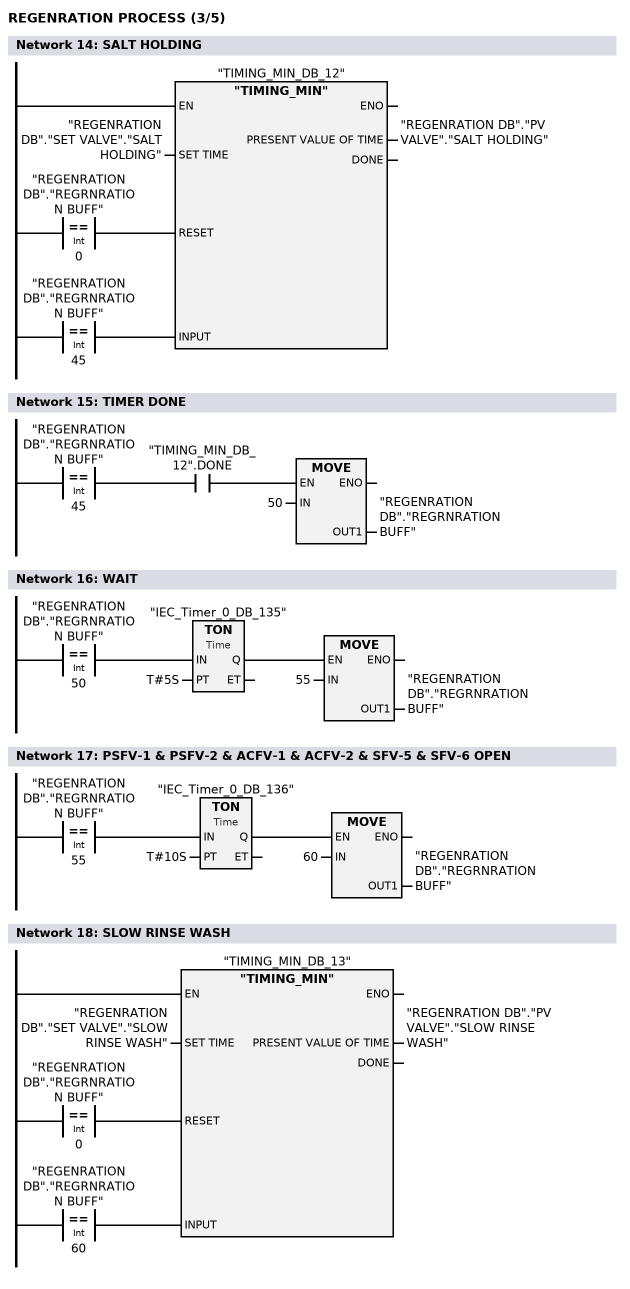
   RUNG wire#powerrail
      "TIMING_MIN_DB_12"(RESET := wire#w1, INPUT := wire#w2, "SET TIME" := "REGENRATION DB"."SET VALVE"."SALT HOLDING", "PRESENT VALUE OF TIME" => "REGENRATION DB"."PV VALVE"."SALT HOLDING", DONE =>)
   END_RUNG
   RUNG wire#powerrail
      { S7_Templates := "SrcType := Int" } EQ_Contact(in1 := "REGENRATION DB"."REGRNRATION BUFF", in2 := 0)
   END_RUNG wire#w1
   RUNG wire#powerrail
      { S7_Templates := "SrcType := Int" } EQ_Contact(in1 := "REGENRATION DB"."REGRNRATION BUFF", in2 := 45)
   END_RUNG wire#w2
   // the same network as SCL:
   "TIMING_MIN_DB_12"("SET TIME" := "REGENRATION DB"."SET VALVE"."SALT HOLDING",   // "TIMING_MIN"
                      RESET := "REGENRATION DB"."REGRNRATION BUFF" = 0,
                      INPUT := "REGENRATION DB"."REGRNRATION BUFF" = 45,
                      "PRESENT VALUE OF TIME" => "REGENRATION DB"."PV VALVE"."SALT HOLDING");
END_REGION

REGION Network 15: TIMER DONE
   RUNG wire#powerrail
      { S7_Templates := "SrcType := Int" } EQ_Contact(in1 := "REGENRATION DB"."REGRNRATION BUFF", in2 := 45)
      Contact( "TIMING_MIN_DB_12".DONE )
      Move(in := 50, out1 => "REGENRATION DB"."REGRNRATION BUFF")
   END_RUNG
   // the same network as SCL:
   IF ("REGENRATION DB"."REGRNRATION BUFF" = 45) AND "TIMING_MIN_DB_12".DONE THEN
       "REGENRATION DB"."REGRNRATION BUFF" := 50;
   END_IF;
END_REGION

REGION Network 16: WAIT
   RUNG wire#powerrail
      { S7_Templates := "SrcType := Int" } EQ_Contact(in1 := "REGENRATION DB"."REGRNRATION BUFF", in2 := 50)
      { S7_Templates := "time_type := Time" } "IEC_Timer_0_DB_135".TON(pt := T#5S, et =>)
      Move(in := 55, out1 => "REGENRATION DB"."REGRNRATION BUFF")
   END_RUNG
   // the same network as SCL:
   "IEC_Timer_0_DB_135".TON(IN := "REGENRATION DB"."REGRNRATION BUFF" = 50, PT := T#5S);
   IF "IEC_Timer_0_DB_135".Q THEN "REGENRATION DB"."REGRNRATION BUFF" := 55; END_IF;
END_REGION

REGION Network 17: PSFV-1 & PSFV-2 & ACFV-1 & ACFV-2 & SFV-5 & SFV-6 OPEN
   RUNG wire#powerrail
      { S7_Templates := "SrcType := Int" } EQ_Contact(in1 := "REGENRATION DB"."REGRNRATION BUFF", in2 := 55)
      { S7_Templates := "time_type := Time" } "IEC_Timer_0_DB_136".TON(pt := T#10S, et =>)
      Move(in := 60, out1 => "REGENRATION DB"."REGRNRATION BUFF")
   END_RUNG
   // the same network as SCL:
   "IEC_Timer_0_DB_136".TON(IN := "REGENRATION DB"."REGRNRATION BUFF" = 55, PT := T#10S);
   IF "IEC_Timer_0_DB_136".Q THEN "REGENRATION DB"."REGRNRATION BUFF" := 60; END_IF;
END_REGION

REGION Network 18: SLOW RINSE WASH
   RUNG wire#powerrail
      "TIMING_MIN_DB_13"(RESET := wire#w1, INPUT := wire#w2, "SET TIME" := "REGENRATION DB"."SET VALVE"."SLOW RINSE WASH", "PRESENT VALUE OF TIME" => "REGENRATION DB"."PV VALVE"."SLOW RINSE WASH", DONE =>)
   END_RUNG
   RUNG wire#powerrail
      { S7_Templates := "SrcType := Int" } EQ_Contact(in1 := "REGENRATION DB"."REGRNRATION BUFF", in2 := 0)
   END_RUNG wire#w1
   RUNG wire#powerrail
      { S7_Templates := "SrcType := Int" } EQ_Contact(in1 := "REGENRATION DB"."REGRNRATION BUFF", in2 := 60)
   END_RUNG wire#w2
   // the same network as SCL:
   "TIMING_MIN_DB_13"("SET TIME" := "REGENRATION DB"."SET VALVE"."SLOW RINSE WASH",   // "TIMING_MIN"
                      RESET := "REGENRATION DB"."REGRNRATION BUFF" = 0,
                      INPUT := "REGENRATION DB"."REGRNRATION BUFF" = 60,
                      "PRESENT VALUE OF TIME" => "REGENRATION DB"."PV VALVE"."SLOW RINSE WASH");
END_REGION

REGION Network 19: TIMER DONE
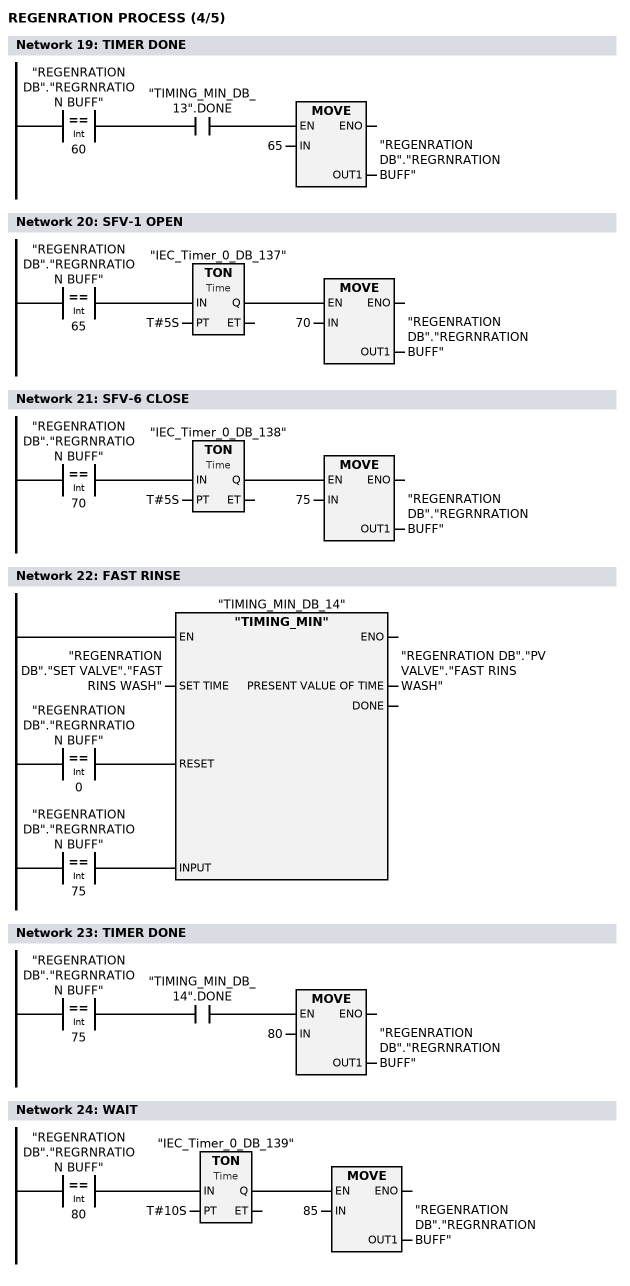
   RUNG wire#powerrail
      { S7_Templates := "SrcType := Int" } EQ_Contact(in1 := "REGENRATION DB"."REGRNRATION BUFF", in2 := 60)
      Contact( "TIMING_MIN_DB_13".DONE )
      Move(in := 65, out1 => "REGENRATION DB"."REGRNRATION BUFF")
   END_RUNG
   // the same network as SCL:
   IF ("REGENRATION DB"."REGRNRATION BUFF" = 60) AND "TIMING_MIN_DB_13".DONE THEN
       "REGENRATION DB"."REGRNRATION BUFF" := 65;
   END_IF;
END_REGION

REGION Network 20: SFV-1 OPEN
   RUNG wire#powerrail
      { S7_Templates := "SrcType := Int" } EQ_Contact(in1 := "REGENRATION DB"."REGRNRATION BUFF", in2 := 65)
      { S7_Templates := "time_type := Time" } "IEC_Timer_0_DB_137".TON(pt := T#5S, et =>)
      Move(in := 70, out1 => "REGENRATION DB"."REGRNRATION BUFF")
   END_RUNG
   // the same network as SCL:
   "IEC_Timer_0_DB_137".TON(IN := "REGENRATION DB"."REGRNRATION BUFF" = 65, PT := T#5S);
   IF "IEC_Timer_0_DB_137".Q THEN "REGENRATION DB"."REGRNRATION BUFF" := 70; END_IF;
END_REGION

REGION Network 21: SFV-6 CLOSE
   RUNG wire#powerrail
      { S7_Templates := "SrcType := Int" } EQ_Contact(in1 := "REGENRATION DB"."REGRNRATION BUFF", in2 := 70)
      { S7_Templates := "time_type := Time" } "IEC_Timer_0_DB_138".TON(pt := T#5S, et =>)
      Move(in := 75, out1 => "REGENRATION DB"."REGRNRATION BUFF")
   END_RUNG
   // the same network as SCL:
   "IEC_Timer_0_DB_138".TON(IN := "REGENRATION DB"."REGRNRATION BUFF" = 70, PT := T#5S);
   IF "IEC_Timer_0_DB_138".Q THEN "REGENRATION DB"."REGRNRATION BUFF" := 75; END_IF;
END_REGION

REGION Network 22: FAST RINSE
   RUNG wire#powerrail
      "TIMING_MIN_DB_14"(RESET := wire#w1, INPUT := wire#w2, "SET TIME" := "REGENRATION DB"."SET VALVE"."FAST RINS WASH", "PRESENT VALUE OF TIME" => "REGENRATION DB"."PV VALVE"."FAST RINS WASH", DONE =>)
   END_RUNG
   RUNG wire#powerrail
      { S7_Templates := "SrcType := Int" } EQ_Contact(in1 := "REGENRATION DB"."REGRNRATION BUFF", in2 := 0)
   END_RUNG wire#w1
   RUNG wire#powerrail
      { S7_Templates := "SrcType := Int" } EQ_Contact(in1 := "REGENRATION DB"."REGRNRATION BUFF", in2 := 75)
   END_RUNG wire#w2
   // the same network as SCL:
   "TIMING_MIN_DB_14"("SET TIME" := "REGENRATION DB"."SET VALVE"."FAST RINS WASH",   // "TIMING_MIN"
                      RESET := "REGENRATION DB"."REGRNRATION BUFF" = 0,
                      INPUT := "REGENRATION DB"."REGRNRATION BUFF" = 75,
                      "PRESENT VALUE OF TIME" => "REGENRATION DB"."PV VALVE"."FAST RINS WASH");
END_REGION

REGION Network 23: TIMER DONE
   RUNG wire#powerrail
      { S7_Templates := "SrcType := Int" } EQ_Contact(in1 := "REGENRATION DB"."REGRNRATION BUFF", in2 := 75)
      Contact( "TIMING_MIN_DB_14".DONE )
      Move(in := 80, out1 => "REGENRATION DB"."REGRNRATION BUFF")
   END_RUNG
   // the same network as SCL:
   IF ("REGENRATION DB"."REGRNRATION BUFF" = 75) AND "TIMING_MIN_DB_14".DONE THEN
       "REGENRATION DB"."REGRNRATION BUFF" := 80;
   END_IF;
END_REGION

REGION Network 24: WAIT
   RUNG wire#powerrail
      { S7_Templates := "SrcType := Int" } EQ_Contact(in1 := "REGENRATION DB"."REGRNRATION BUFF", in2 := 80)
      { S7_Templates := "time_type := Time" } "IEC_Timer_0_DB_139".TON(pt := T#10S, et =>)
      Move(in := 85, out1 => "REGENRATION DB"."REGRNRATION BUFF")
   END_RUNG
   // the same network as SCL:
   "IEC_Timer_0_DB_139".TON(IN := "REGENRATION DB"."REGRNRATION BUFF" = 80, PT := T#10S);
   IF "IEC_Timer_0_DB_139".Q THEN "REGENRATION DB"."REGRNRATION BUFF" := 85; END_IF;
END_REGION

REGION Network 25: PSFV-1 & PSFV-2 & ACFV-1 & ACFV-2 & SFV-5 & SFV-1 CLOSE
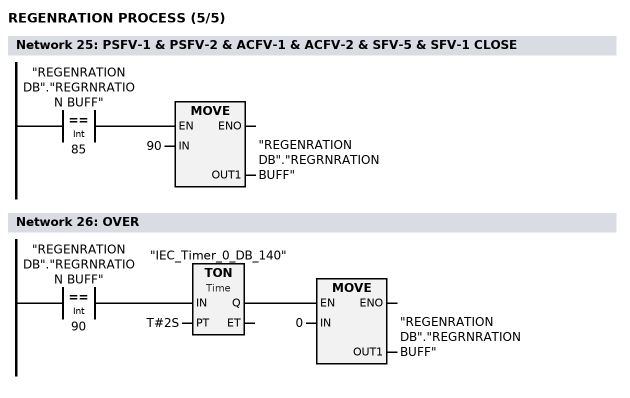
   RUNG wire#powerrail
      { S7_Templates := "SrcType := Int" } EQ_Contact(in1 := "REGENRATION DB"."REGRNRATION BUFF", in2 := 85)
      Move(in := 90, out1 => "REGENRATION DB"."REGRNRATION BUFF")
   END_RUNG
   // the same network as SCL:
   IF "REGENRATION DB"."REGRNRATION BUFF" = 85 THEN "REGENRATION DB"."REGRNRATION BUFF" := 90; END_IF;
END_REGION

REGION Network 26: OVER
   RUNG wire#powerrail
      { S7_Templates := "SrcType := Int" } EQ_Contact(in1 := "REGENRATION DB"."REGRNRATION BUFF", in2 := 90)
      { S7_Templates := "time_type := Time" } "IEC_Timer_0_DB_140".TON(pt := T#2S, et =>)
      Move(in := 0, out1 => "REGENRATION DB"."REGRNRATION BUFF")
   END_RUNG
   // the same network as SCL:
   "IEC_Timer_0_DB_140".TON(IN := "REGENRATION DB"."REGRNRATION BUFF" = 90, PT := T#2S);
   IF "IEC_Timer_0_DB_140".Q THEN "REGENRATION DB"."REGRNRATION BUFF" := 0; END_IF;
END_REGION
END_FUNCTION

FUNCTION "RO PROCESS." : Void   // FC15, LAD
{ S7_Optimized_Access := 'TRUE' }
// stored: SetENOAutomatically false
BEGIN

REGION Network 1: AUTO FLUSHING AV3
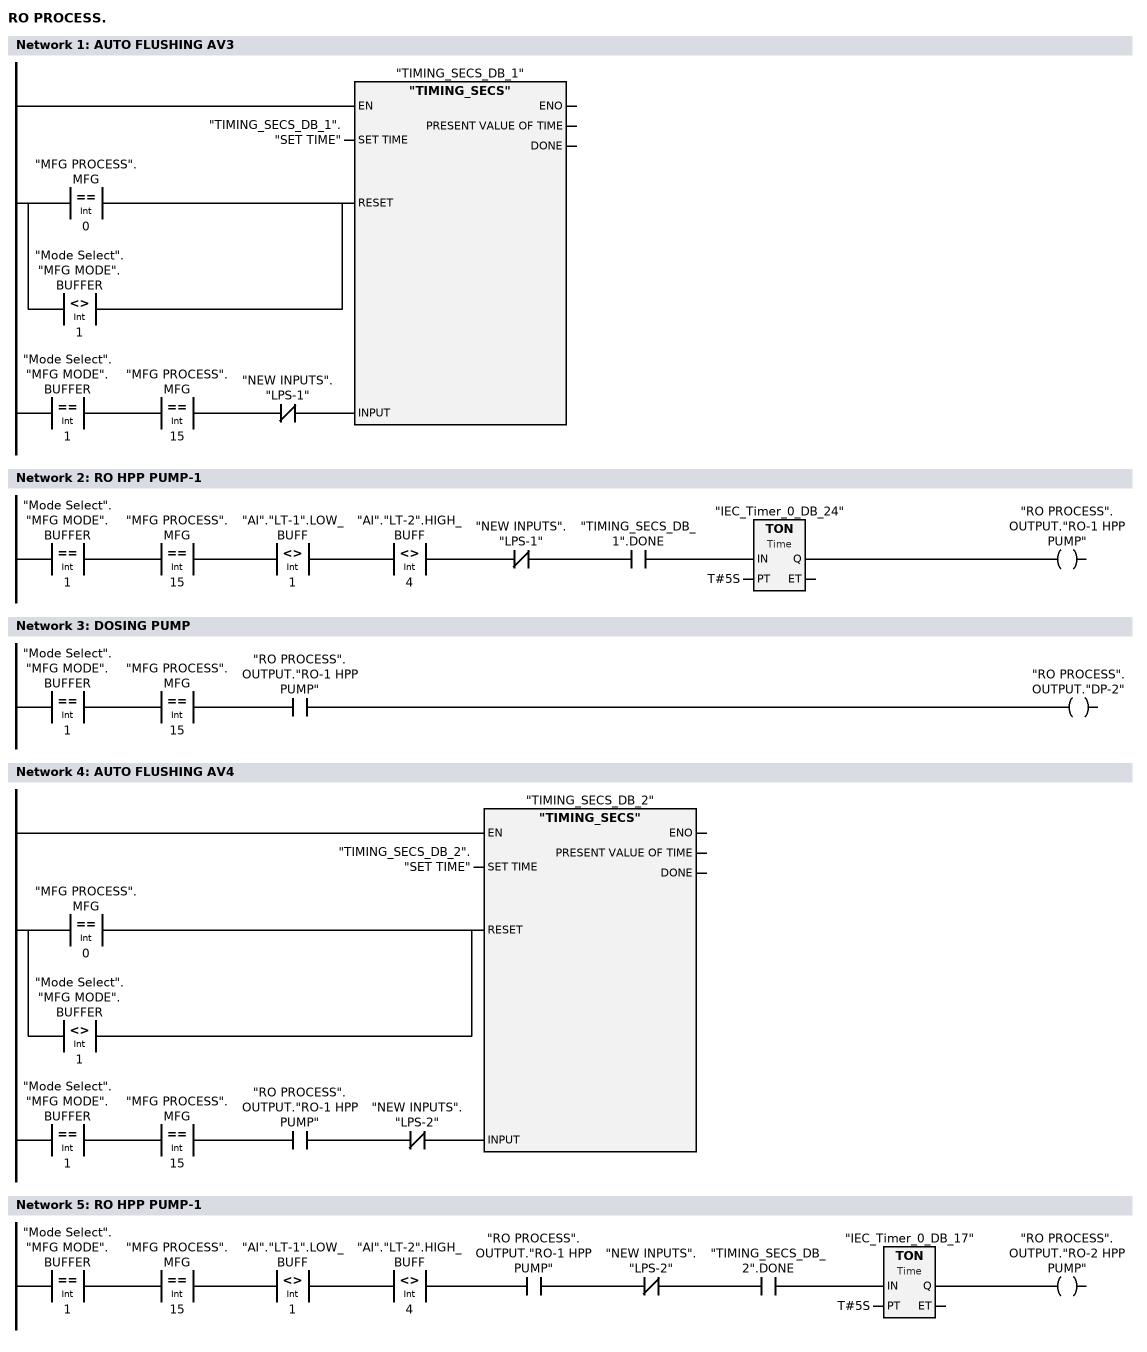
   RUNG wire#powerrail
      "TIMING_SECS_DB_1"(RESET := wire#w1, INPUT := wire#w2, "SET TIME" := "TIMING_SECS_DB_1"."SET TIME", "PRESENT VALUE OF TIME" =>, DONE =>)
   END_RUNG
   RUNG wire#powerrail
      { S7_Templates := "SrcType := Int" } EQ_Contact(in1 := "MFG PROCESS".MFG, in2 := 0)
   END_RUNG wire#w1
   RUNG wire#powerrail
      { S7_Templates := "SrcType := Int" } NE_Contact(in1 := "Mode Select"."MFG MODE".BUFFER, in2 := 1)
   END_RUNG wire#w1
   RUNG wire#powerrail
      { S7_Templates := "SrcType := Int" } EQ_Contact(in1 := "Mode Select"."MFG MODE".BUFFER, in2 := 1)
      { S7_Templates := "SrcType := Int" } EQ_Contact(in1 := "MFG PROCESS".MFG, in2 := 15)
      I_Contact( "NEW INPUTS"."LPS-1" )
   END_RUNG wire#w2
   // the same network as SCL:
   "TIMING_SECS_DB_1"("SET TIME" := "TIMING_SECS_DB_1"."SET TIME",   // "TIMING_SECS"
                      RESET := ("MFG PROCESS".MFG = 0) OR ("Mode Select"."MFG MODE".BUFFER <> 1),
                      INPUT := ("Mode Select"."MFG MODE".BUFFER = 1) AND ("MFG PROCESS".MFG = 15) AND NOT "NEW INPUTS"."LPS-1");
END_REGION

REGION Network 2: RO HPP PUMP-1
   RUNG wire#powerrail
      { S7_Templates := "SrcType := Int" } EQ_Contact(in1 := "Mode Select"."MFG MODE".BUFFER, in2 := 1)
      { S7_Templates := "SrcType := Int" } EQ_Contact(in1 := "MFG PROCESS".MFG, in2 := 15)
      { S7_Templates := "SrcType := Int" } NE_Contact(in1 := "AI"."LT-1".LOW_BUFF, in2 := 1)
      { S7_Templates := "SrcType := Int" } NE_Contact(in1 := "AI"."LT-2".HIGH_BUFF, in2 := 4)
      I_Contact( "NEW INPUTS"."LPS-1" )
      Contact( "TIMING_SECS_DB_1".DONE )
      { S7_Templates := "time_type := Time" } "IEC_Timer_0_DB_24".TON(pt := T#5S, et =>)
      Coil( "RO PROCESS".OUTPUT."RO-1 HPP PUMP" )
   END_RUNG
   // the same network as SCL:
   "IEC_Timer_0_DB_24".TON(IN := ("Mode Select"."MFG MODE".BUFFER = 1) AND ("MFG PROCESS".MFG = 15) AND ("AI"."LT-1".LOW_BUFF <> 1) AND ("AI"."LT-2".HIGH_BUFF <> 4) AND NOT "NEW INPUTS"."LPS-1" AND "TIMING_SECS_DB_1".DONE,
                           PT := T#5S);
   "RO PROCESS".OUTPUT."RO-1 HPP PUMP" := "IEC_Timer_0_DB_24".Q;
END_REGION

REGION Network 3: DOSING PUMP
   RUNG wire#powerrail
      { S7_Templates := "SrcType := Int" } EQ_Contact(in1 := "Mode Select"."MFG MODE".BUFFER, in2 := 1)
      { S7_Templates := "SrcType := Int" } EQ_Contact(in1 := "MFG PROCESS".MFG, in2 := 15)
      Contact( "RO PROCESS".OUTPUT."RO-1 HPP PUMP" )
      Coil( "RO PROCESS".OUTPUT."DP-2" )
   END_RUNG
   // the same network as SCL:
   "RO PROCESS".OUTPUT."DP-2" := ("Mode Select"."MFG MODE".BUFFER = 1) AND ("MFG PROCESS".MFG = 15) AND "RO PROCESS".OUTPUT."RO-1 HPP PUMP";
END_REGION

REGION Network 4: AUTO FLUSHING AV4
   RUNG wire#powerrail
      "TIMING_SECS_DB_2"(RESET := wire#w1, INPUT := wire#w2, "SET TIME" := "TIMING_SECS_DB_2"."SET TIME", "PRESENT VALUE OF TIME" =>, DONE =>)
   END_RUNG
   RUNG wire#powerrail
      { S7_Templates := "SrcType := Int" } EQ_Contact(in1 := "MFG PROCESS".MFG, in2 := 0)
   END_RUNG wire#w1
   RUNG wire#powerrail
      { S7_Templates := "SrcType := Int" } NE_Contact(in1 := "Mode Select"."MFG MODE".BUFFER, in2 := 1)
   END_RUNG wire#w1
   RUNG wire#powerrail
      { S7_Templates := "SrcType := Int" } EQ_Contact(in1 := "Mode Select"."MFG MODE".BUFFER, in2 := 1)
      { S7_Templates := "SrcType := Int" } EQ_Contact(in1 := "MFG PROCESS".MFG, in2 := 15)
      Contact( "RO PROCESS".OUTPUT."RO-1 HPP PUMP" )
      I_Contact( "NEW INPUTS"."LPS-2" )
   END_RUNG wire#w2
   // the same network as SCL:
   "TIMING_SECS_DB_2"("SET TIME" := "TIMING_SECS_DB_2"."SET TIME",   // "TIMING_SECS"
                      RESET := ("MFG PROCESS".MFG = 0) OR ("Mode Select"."MFG MODE".BUFFER <> 1),
                      INPUT := ("Mode Select"."MFG MODE".BUFFER = 1) AND ("MFG PROCESS".MFG = 15) AND "RO PROCESS".OUTPUT."RO-1 HPP PUMP" AND NOT "NEW INPUTS"."LPS-2");
END_REGION

REGION Network 5: RO HPP PUMP-1
   RUNG wire#powerrail
      { S7_Templates := "SrcType := Int" } EQ_Contact(in1 := "Mode Select"."MFG MODE".BUFFER, in2 := 1)
      { S7_Templates := "SrcType := Int" } EQ_Contact(in1 := "MFG PROCESS".MFG, in2 := 15)
      { S7_Templates := "SrcType := Int" } NE_Contact(in1 := "AI"."LT-1".LOW_BUFF, in2 := 1)
      { S7_Templates := "SrcType := Int" } NE_Contact(in1 := "AI"."LT-2".HIGH_BUFF, in2 := 4)
      Contact( "RO PROCESS".OUTPUT."RO-1 HPP PUMP" )
      I_Contact( "NEW INPUTS"."LPS-2" )
      Contact( "TIMING_SECS_DB_2".DONE )
      { S7_Templates := "time_type := Time" } "IEC_Timer_0_DB_17".TON(pt := T#5S, et =>)
      Coil( "RO PROCESS".OUTPUT."RO-2 HPP PUMP" )
   END_RUNG
   // the same network as SCL:
   "IEC_Timer_0_DB_17".TON(IN := ("Mode Select"."MFG MODE".BUFFER = 1) AND ("MFG PROCESS".MFG = 15) AND ("AI"."LT-1".LOW_BUFF <> 1) AND ("AI"."LT-2".HIGH_BUFF <> 4) AND "RO PROCESS".OUTPUT."RO-1 HPP PUMP" AND NOT "NEW INPUTS"."LPS-2" AND "TIMING_SECS_DB_2".DONE,
                           PT := T#5S);
   "RO PROCESS".OUTPUT."RO-2 HPP PUMP" := "IEC_Timer_0_DB_17".Q;
END_REGION
END_FUNCTION

FUNCTION_BLOCK "TIMING_SECS"   // FB1, LAD
{ S7_Optimized_Access := 'TRUE' }
// stored: MemoryReserve 100, SetENOAutomatically false
   VAR_INPUT
      "SET TIME" : Int;
      RESET : Bool;
      INPUT : Bool;
   END_VAR
   VAR_OUTPUT
      "PRESENT VALUE OF TIME" : Int;
      DONE : Bool;
   END_VAR
   VAR
      "TIMER 1" { S7_SetPoint := 'True'} : IEC_TIMER;
   END_VAR
   VAR RETAIN
      "COUNTER1 1" { S7_SetPoint := 'True'} : IEC_COUNTER;
   END_VAR
   VAR_TEMP   // added for the SCL form of the ladder/FBD networks
      _w1 : Bool;
      _w2 : Bool;
   END_VAR
BEGIN

REGION Network 1
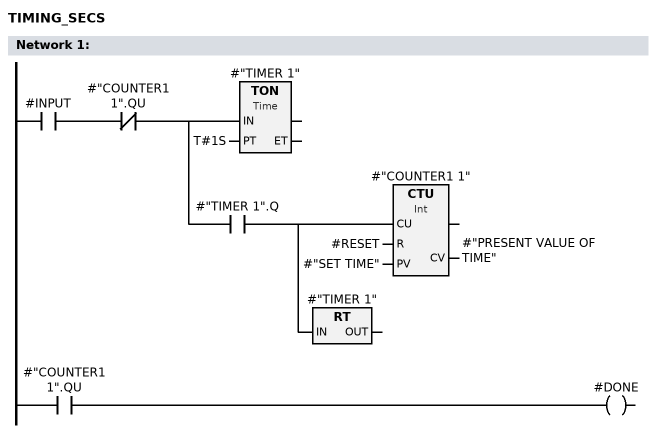
   RUNG wire#powerrail
      Contact( #INPUT )
      I_Contact( #"COUNTER1 1".QU )
      wire#w1
      { S7_Templates := "time_type := Time" } #"TIMER 1".TON(pt := T#1S, et =>)
   END_RUNG
   RUNG wire#w1
      Contact( #"TIMER 1".Q )
      wire#w2
      { S7_Templates := "value_type := Int" } #"COUNTER1 1".CTU(r := #RESET, pv := #"SET TIME", cv => #"PRESENT VALUE OF TIME")
   END_RUNG
   RUNG wire#w2
      RT_Coil( #"TIMER 1" )
   END_RUNG
   RUNG wire#powerrail
      Contact( #"COUNTER1 1".QU )
      Coil( #DONE )
   END_RUNG
   // the same network as SCL:
   #_w1 := #INPUT AND NOT #"COUNTER1 1".QU;
   #"TIMER 1".TON(IN := #_w1, PT := T#1S);
   #_w2 := #_w1 AND #"TIMER 1".Q;
   #"COUNTER1 1".CTU(CU := #_w2, R := #RESET, PV := #"SET TIME", CV => #"PRESENT VALUE OF TIME");
   IF #_w2 THEN RESET_TIMER(#"TIMER 1"); END_IF;
   #DONE := #"COUNTER1 1".QU;
END_REGION
END_FUNCTION_BLOCK

FUNCTION_BLOCK "SCALE AO"   // FB5, LAD
{ S7_Optimized_Access := 'TRUE' }
// stored: MemoryReserve 100, SetENOAutomatically false
   VAR_INPUT
      "SET RPM" : Real;
      "MIN RPM" : Real;
      "MAX RPM" : Real;
      "MIN RAW" : Int;
      "MAX RAW" : Int;
   END_VAR
   VAR_OUTPUT
      MODBUS : Int;
   END_VAR
   VAR_TEMP
      NOM : Real;
   END_VAR
BEGIN

REGION Network 1
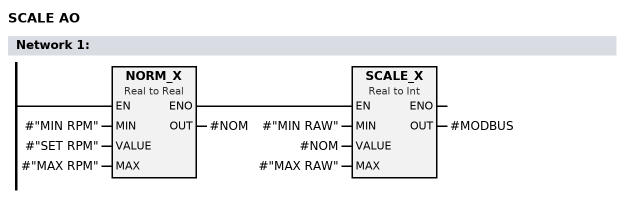
   RUNG wire#powerrail
      { S7_Templates := "[SrcType := Real, DestType := Real]" } Normalize(min := #"MIN RPM", value := #"SET RPM", max := #"MAX RPM", out => #NOM)
      { S7_Templates := "[SrcType := Real, DestType := Int]" } Scale(min := #"MIN RAW", value := #NOM, max := #"MAX RAW", out => #MODBUS)
   END_RUNG
   // the same network as SCL:
   #NOM := NORM_X(MIN := #"MIN RPM", VALUE := #"SET RPM", MAX := #"MAX RPM");
   #MODBUS := SCALE_X(MIN := #"MIN RAW", VALUE := #NOM, MAX := #"MAX RAW");
END_REGION
END_FUNCTION_BLOCK

DATA_BLOCK "SCALE_DB"   // DB9
// stored: InstanceOfName SCALE, InstanceOfType FB
"SCALE"
BEGIN
END_DATA_BLOCK

DATA_BLOCK "SCALE_DB_1"   // DB10
// stored: InstanceOfName SCALE, InstanceOfType FB
"SCALE"
BEGIN
END_DATA_BLOCK

DATA_BLOCK "SCALE_DB_2"   // DB17
// stored: InstanceOfName SCALE, InstanceOfType FB
"SCALE"
BEGIN
END_DATA_BLOCK

DATA_BLOCK "SCALE_DB_3"   // DB19
// stored: InstanceOfName SCALE, InstanceOfType FB
"SCALE"
BEGIN
END_DATA_BLOCK

DATA_BLOCK "HOUR_DB_2"   // DB22
// stored: InstanceOfName HOUR, InstanceOfType FB
"HOUR"
BEGIN
END_DATA_BLOCK

DATA_BLOCK "HOUR_DB_3"   // DB56
// stored: InstanceOfName HOUR, InstanceOfType FB
"HOUR"
BEGIN
END_DATA_BLOCK

DATA_BLOCK "TIMING_MIN_DB"   // DB29
// stored: InstanceOfName TIMING_MIN, InstanceOfType FB
"TIMING_MIN"
BEGIN
END_DATA_BLOCK

DATA_BLOCK "TIMING_MIN_DB_1"   // DB34
// stored: InstanceOfName TIMING_MIN, InstanceOfType FB
"TIMING_MIN"
BEGIN
END_DATA_BLOCK

DATA_BLOCK "TIMING_MIN_DB_15"   // DB23
// stored: InstanceOfName TIMING_MIN, InstanceOfType FB
"TIMING_MIN"
BEGIN
END_DATA_BLOCK

DATA_BLOCK "TIMING_MIN_DB_2"   // DB37
// stored: InstanceOfName TIMING_MIN, InstanceOfType FB
"TIMING_MIN"
BEGIN
END_DATA_BLOCK

DATA_BLOCK "TIMING_MIN_DB_3"   // DB41
// stored: InstanceOfName TIMING_MIN, InstanceOfType FB
"TIMING_MIN"
BEGIN
END_DATA_BLOCK

DATA_BLOCK "TIMING_MIN_DB_4"   // DB50
// stored: InstanceOfName TIMING_MIN, InstanceOfType FB
"TIMING_MIN"
BEGIN
END_DATA_BLOCK

DATA_BLOCK "TIMING_MIN_DB_5"   // DB55
// stored: InstanceOfName TIMING_MIN, InstanceOfType FB
"TIMING_MIN"
BEGIN
END_DATA_BLOCK

DATA_BLOCK "TIMING_MIN_DB_6"   // DB60
// stored: InstanceOfName TIMING_MIN, InstanceOfType FB
"TIMING_MIN"
BEGIN
END_DATA_BLOCK

DATA_BLOCK "TIMING_MIN_DB_7"   // DB66
// stored: InstanceOfName TIMING_MIN, InstanceOfType FB
"TIMING_MIN"
BEGIN
END_DATA_BLOCK

DATA_BLOCK "TIMING_MIN_DB_8"   // DB69
// stored: InstanceOfName TIMING_MIN, InstanceOfType FB
"TIMING_MIN"
BEGIN
END_DATA_BLOCK

DATA_BLOCK "TIMING_MIN_DB_9"   // DB75
// stored: InstanceOfName TIMING_MIN, InstanceOfType FB
"TIMING_MIN"
BEGIN
END_DATA_BLOCK

DATA_BLOCK "TIMING_SECS_DB_1"   // DB42
// stored: InstanceOfName TIMING_SECS, InstanceOfType FB
"TIMING_SECS"
BEGIN
END_DATA_BLOCK

DATA_BLOCK "TIMING_SECS_DB_2"   // DB47
// stored: InstanceOfName TIMING_SECS, InstanceOfType FB
"TIMING_SECS"
BEGIN
END_DATA_BLOCK

DATA_BLOCK "TIMING_MIN_DB_10"   // DB89
// stored: InstanceOfName TIMING_MIN, InstanceOfType FB
"TIMING_MIN"
BEGIN
END_DATA_BLOCK

DATA_BLOCK "TIMING_MIN_DB_11"   // DB108
// stored: InstanceOfName TIMING_MIN, InstanceOfType FB
"TIMING_MIN"
BEGIN
END_DATA_BLOCK

DATA_BLOCK "TIMING_MIN_DB_12"   // DB110
// stored: InstanceOfName TIMING_MIN, InstanceOfType FB
"TIMING_MIN"
BEGIN
END_DATA_BLOCK

DATA_BLOCK "TIMING_MIN_DB_13"   // DB174
// stored: InstanceOfName TIMING_MIN, InstanceOfType FB
"TIMING_MIN"
BEGIN
END_DATA_BLOCK

DATA_BLOCK "TIMING_MIN_DB_14"   // DB177
// stored: InstanceOfName TIMING_MIN, InstanceOfType FB
"TIMING_MIN"
BEGIN
END_DATA_BLOCK

DATA_BLOCK "IEC_Timer_0_DB"   // DB13
{ S7_Optimized_Access := 'TRUE' }
// stored: InstanceOfName IEC_TIMER, OfSystemLibElement IEC_TIMER, OfSystemLibVersion 1.0
"IEC_TIMER"
   // VAR
   //    PT : Time;
   //    ET { ExternalWritable := 'False'} : Time;
   //    IN : Bool;
   //    Q { ExternalWritable := 'False'} : Bool;
   // END_VAR
BEGIN
END_DATA_BLOCK

DATA_BLOCK "IEC_Timer_0_DB_1"   // DB15
{ S7_Optimized_Access := 'TRUE' }
// stored: InstanceOfName IEC_TIMER, OfSystemLibElement IEC_TIMER, OfSystemLibVersion 1.0
"IEC_TIMER"
   // VAR
   //    PT : Time;
   //    ET { ExternalWritable := 'False'} : Time;
   //    IN : Bool;
   //    Q { ExternalWritable := 'False'} : Bool;
   // END_VAR
BEGIN
END_DATA_BLOCK

DATA_BLOCK "IEC_Timer_0_DB_10"   // DB27
{ S7_Optimized_Access := 'TRUE' }
// stored: InstanceOfName IEC_TIMER, OfSystemLibElement IEC_TIMER, OfSystemLibVersion 1.0
"IEC_TIMER"
   // VAR
   //    PT : Time;
   //    ET { ExternalWritable := 'False'} : Time;
   //    IN : Bool;
   //    Q { ExternalWritable := 'False'} : Bool;
   // END_VAR
BEGIN
END_DATA_BLOCK

DATA_BLOCK "IEC_Timer_0_DB_11"   // DB48
{ S7_Optimized_Access := 'TRUE' }
// stored: InstanceOfName IEC_TIMER, OfSystemLibElement IEC_TIMER, OfSystemLibVersion 1.0
"IEC_TIMER"
   // VAR
   //    PT : Time;
   //    ET { ExternalWritable := 'False'} : Time;
   //    IN : Bool;
   //    Q { ExternalWritable := 'False'} : Bool;
   // END_VAR
BEGIN
END_DATA_BLOCK

DATA_BLOCK "IEC_Timer_0_DB_12"   // DB30
{ S7_Optimized_Access := 'TRUE' }
// stored: InstanceOfName IEC_TIMER, OfSystemLibElement IEC_TIMER, OfSystemLibVersion 1.0
"IEC_TIMER"
   // VAR
   //    PT : Time;
   //    ET { ExternalWritable := 'False'} : Time;
   //    IN : Bool;
   //    Q { ExternalWritable := 'False'} : Bool;
   // END_VAR
BEGIN
END_DATA_BLOCK

DATA_BLOCK "IEC_Timer_0_DB_129"   // DB167
{ S7_Optimized_Access := 'TRUE' }
// stored: InstanceOfName IEC_TIMER, OfSystemLibElement IEC_TIMER, OfSystemLibVersion 1.0
"IEC_TIMER"
   // VAR
   //    PT : Time;
   //    ET { ExternalWritable := 'False'} : Time;
   //    IN : Bool;
   //    Q { ExternalWritable := 'False'} : Bool;
   // END_VAR
BEGIN
END_DATA_BLOCK

DATA_BLOCK "IEC_Timer_0_DB_13"   // DB31
{ S7_Optimized_Access := 'TRUE' }
// stored: InstanceOfName IEC_TIMER, OfSystemLibElement IEC_TIMER, OfSystemLibVersion 1.0
"IEC_TIMER"
   // VAR
   //    PT : Time;
   //    ET { ExternalWritable := 'False'} : Time;
   //    IN : Bool;
   //    Q { ExternalWritable := 'False'} : Bool;
   // END_VAR
BEGIN
END_DATA_BLOCK

DATA_BLOCK "IEC_Timer_0_DB_132"   // DB171
{ S7_Optimized_Access := 'TRUE' }
// stored: InstanceOfName IEC_TIMER, OfSystemLibElement IEC_TIMER, OfSystemLibVersion 1.0
"IEC_TIMER"
   // VAR
   //    PT : Time;
   //    ET { ExternalWritable := 'False'} : Time;
   //    IN : Bool;
   //    Q { ExternalWritable := 'False'} : Bool;
   // END_VAR
BEGIN
END_DATA_BLOCK

DATA_BLOCK "IEC_Timer_0_DB_133"   // DB172
{ S7_Optimized_Access := 'TRUE' }
// stored: InstanceOfName IEC_TIMER, OfSystemLibElement IEC_TIMER, OfSystemLibVersion 1.0
"IEC_TIMER"
   // VAR
   //    PT : Time;
   //    ET { ExternalWritable := 'False'} : Time;
   //    IN : Bool;
   //    Q { ExternalWritable := 'False'} : Bool;
   // END_VAR
BEGIN
END_DATA_BLOCK

DATA_BLOCK "IEC_Timer_0_DB_135"   // DB111
{ S7_Optimized_Access := 'TRUE' }
// stored: InstanceOfName IEC_TIMER, OfSystemLibElement IEC_TIMER, OfSystemLibVersion 1.0
"IEC_TIMER"
   // VAR
   //    PT : Time;
   //    ET { ExternalWritable := 'False'} : Time;
   //    IN : Bool;
   //    Q { ExternalWritable := 'False'} : Bool;
   // END_VAR
BEGIN
END_DATA_BLOCK

DATA_BLOCK "IEC_Timer_0_DB_136"   // DB112
{ S7_Optimized_Access := 'TRUE' }
// stored: InstanceOfName IEC_TIMER, OfSystemLibElement IEC_TIMER, OfSystemLibVersion 1.0
"IEC_TIMER"
   // VAR
   //    PT : Time;
   //    ET { ExternalWritable := 'False'} : Time;
   //    IN : Bool;
   //    Q { ExternalWritable := 'False'} : Bool;
   // END_VAR
BEGIN
END_DATA_BLOCK

DATA_BLOCK "IEC_Timer_0_DB_137"   // DB175
{ S7_Optimized_Access := 'TRUE' }
// stored: InstanceOfName IEC_TIMER, OfSystemLibElement IEC_TIMER, OfSystemLibVersion 1.0
"IEC_TIMER"
   // VAR
   //    PT : Time;
   //    ET { ExternalWritable := 'False'} : Time;
   //    IN : Bool;
   //    Q { ExternalWritable := 'False'} : Bool;
   // END_VAR
BEGIN
END_DATA_BLOCK

DATA_BLOCK "IEC_Timer_0_DB_138"   // DB176
{ S7_Optimized_Access := 'TRUE' }
// stored: InstanceOfName IEC_TIMER, OfSystemLibElement IEC_TIMER, OfSystemLibVersion 1.0
"IEC_TIMER"
   // VAR
   //    PT : Time;
   //    ET { ExternalWritable := 'False'} : Time;
   //    IN : Bool;
   //    Q { ExternalWritable := 'False'} : Bool;
   // END_VAR
BEGIN
END_DATA_BLOCK

DATA_BLOCK "IEC_Timer_0_DB_139"   // DB178
{ S7_Optimized_Access := 'TRUE' }
// stored: InstanceOfName IEC_TIMER, OfSystemLibElement IEC_TIMER, OfSystemLibVersion 1.0
"IEC_TIMER"
   // VAR
   //    PT : Time;
   //    ET { ExternalWritable := 'False'} : Time;
   //    IN : Bool;
   //    Q { ExternalWritable := 'False'} : Bool;
   // END_VAR
BEGIN
END_DATA_BLOCK

DATA_BLOCK "IEC_Timer_0_DB_14"   // DB32
{ S7_Optimized_Access := 'TRUE' }
// stored: InstanceOfName IEC_TIMER, OfSystemLibElement IEC_TIMER, OfSystemLibVersion 1.0
"IEC_TIMER"
   // VAR
   //    PT : Time;
   //    ET { ExternalWritable := 'False'} : Time;
   //    IN : Bool;
   //    Q { ExternalWritable := 'False'} : Bool;
   // END_VAR
BEGIN
END_DATA_BLOCK

DATA_BLOCK "IEC_Timer_0_DB_140"   // DB179
{ S7_Optimized_Access := 'TRUE' }
// stored: InstanceOfName IEC_TIMER, OfSystemLibElement IEC_TIMER, OfSystemLibVersion 1.0
"IEC_TIMER"
   // VAR
   //    PT : Time;
   //    ET { ExternalWritable := 'False'} : Time;
   //    IN : Bool;
   //    Q { ExternalWritable := 'False'} : Bool;
   // END_VAR
BEGIN
END_DATA_BLOCK

DATA_BLOCK "IEC_Timer_0_DB_15"   // DB33
{ S7_Optimized_Access := 'TRUE' }
// stored: InstanceOfName IEC_TIMER, OfSystemLibElement IEC_TIMER, OfSystemLibVersion 1.0
"IEC_TIMER"
   // VAR
   //    PT : Time;
   //    ET { ExternalWritable := 'False'} : Time;
   //    IN : Bool;
   //    Q { ExternalWritable := 'False'} : Bool;
   // END_VAR
BEGIN
END_DATA_BLOCK

DATA_BLOCK "IEC_Timer_0_DB_16"   // DB35
{ S7_Optimized_Access := 'TRUE' }
// stored: InstanceOfName IEC_TIMER, OfSystemLibElement IEC_TIMER, OfSystemLibVersion 1.0
"IEC_TIMER"
   // VAR
   //    PT : Time;
   //    ET { ExternalWritable := 'False'} : Time;
   //    IN : Bool;
   //    Q { ExternalWritable := 'False'} : Bool;
   // END_VAR
BEGIN
END_DATA_BLOCK

DATA_BLOCK "IEC_Timer_0_DB_17"   // DB36
{ S7_Optimized_Access := 'TRUE' }
// stored: InstanceOfName IEC_TIMER, OfSystemLibElement IEC_TIMER, OfSystemLibVersion 1.0
"IEC_TIMER"
   // VAR
   //    PT : Time;
   //    ET { ExternalWritable := 'False'} : Time;
   //    IN : Bool;
   //    Q { ExternalWritable := 'False'} : Bool;
   // END_VAR
BEGIN
END_DATA_BLOCK

DATA_BLOCK "IEC_Timer_0_DB_18"   // DB38
{ S7_Optimized_Access := 'TRUE' }
// stored: InstanceOfName IEC_TIMER, OfSystemLibElement IEC_TIMER, OfSystemLibVersion 1.0
"IEC_TIMER"
   // VAR
   //    PT : Time;
   //    ET { ExternalWritable := 'False'} : Time;
   //    IN : Bool;
   //    Q { ExternalWritable := 'False'} : Bool;
   // END_VAR
BEGIN
END_DATA_BLOCK

DATA_BLOCK "IEC_Timer_0_DB_19"   // DB39
{ S7_Optimized_Access := 'TRUE' }
// stored: InstanceOfName IEC_TIMER, OfSystemLibElement IEC_TIMER, OfSystemLibVersion 1.0
"IEC_TIMER"
   // VAR
   //    PT : Time;
   //    ET { ExternalWritable := 'False'} : Time;
   //    IN : Bool;
   //    Q { ExternalWritable := 'False'} : Bool;
   // END_VAR
BEGIN
END_DATA_BLOCK

DATA_BLOCK "IEC_Timer_0_DB_2"   // DB57
{ S7_Optimized_Access := 'TRUE' }
// stored: InstanceOfName IEC_TIMER, OfSystemLibElement IEC_TIMER, OfSystemLibVersion 1.0
"IEC_TIMER"
   // VAR
   //    PT : Time;
   //    ET { ExternalWritable := 'False'} : Time;
   //    IN : Bool;
   //    Q { ExternalWritable := 'False'} : Bool;
   // END_VAR
BEGIN
END_DATA_BLOCK

DATA_BLOCK "IEC_Timer_0_DB_20"   // DB40
{ S7_Optimized_Access := 'TRUE' }
// stored: InstanceOfName IEC_TIMER, OfSystemLibElement IEC_TIMER, OfSystemLibVersion 1.0
"IEC_TIMER"
   // VAR
   //    PT : Time;
   //    ET { ExternalWritable := 'False'} : Time;
   //    IN : Bool;
   //    Q { ExternalWritable := 'False'} : Bool;
   // END_VAR
BEGIN
END_DATA_BLOCK

DATA_BLOCK "IEC_Timer_0_DB_21"   // DB1
{ S7_Optimized_Access := 'TRUE' }
// stored: InstanceOfName IEC_TIMER, OfSystemLibElement IEC_TIMER, OfSystemLibVersion 1.0
"IEC_TIMER"
   // VAR
   //    PT : Time;
   //    ET { ExternalWritable := 'False'} : Time;
   //    IN : Bool;
   //    Q { ExternalWritable := 'False'} : Bool;
   // END_VAR
BEGIN
END_DATA_BLOCK

DATA_BLOCK "IEC_Timer_0_DB_22"   // DB43
{ S7_Optimized_Access := 'TRUE' }
// stored: InstanceOfName IEC_TIMER, OfSystemLibElement IEC_TIMER, OfSystemLibVersion 1.0
"IEC_TIMER"
   // VAR
   //    PT : Time;
   //    ET { ExternalWritable := 'False'} : Time;
   //    IN : Bool;
   //    Q { ExternalWritable := 'False'} : Bool;
   // END_VAR
BEGIN
END_DATA_BLOCK

DATA_BLOCK "IEC_Timer_0_DB_23"   // DB44
{ S7_Optimized_Access := 'TRUE' }
// stored: InstanceOfName IEC_TIMER, OfSystemLibElement IEC_TIMER, OfSystemLibVersion 1.0
"IEC_TIMER"
   // VAR
   //    PT : Time;
   //    ET { ExternalWritable := 'False'} : Time;
   //    IN : Bool;
   //    Q { ExternalWritable := 'False'} : Bool;
   // END_VAR
BEGIN
END_DATA_BLOCK

DATA_BLOCK "IEC_Timer_0_DB_24"   // DB45
{ S7_Optimized_Access := 'TRUE' }
// stored: InstanceOfName IEC_TIMER, OfSystemLibElement IEC_TIMER, OfSystemLibVersion 1.0
"IEC_TIMER"
   // VAR
   //    PT : Time;
   //    ET { ExternalWritable := 'False'} : Time;
   //    IN : Bool;
   //    Q { ExternalWritable := 'False'} : Bool;
   // END_VAR
BEGIN
END_DATA_BLOCK

DATA_BLOCK "IEC_Timer_0_DB_25"   // DB49
{ S7_Optimized_Access := 'TRUE' }
// stored: InstanceOfName IEC_TIMER, OfSystemLibElement IEC_TIMER, OfSystemLibVersion 1.0
"IEC_TIMER"
   // VAR
   //    PT : Time;
   //    ET { ExternalWritable := 'False'} : Time;
   //    IN : Bool;
   //    Q { ExternalWritable := 'False'} : Bool;
   // END_VAR
BEGIN
END_DATA_BLOCK

DATA_BLOCK "IEC_Timer_0_DB_26"   // DB2
{ S7_Optimized_Access := 'TRUE' }
// stored: InstanceOfName IEC_TIMER, OfSystemLibElement IEC_TIMER, OfSystemLibVersion 1.0
"IEC_TIMER"
   // VAR
   //    PT : Time;
   //    ET { ExternalWritable := 'False'} : Time;
   //    IN : Bool;
   //    Q { ExternalWritable := 'False'} : Bool;
   // END_VAR
BEGIN
END_DATA_BLOCK

DATA_BLOCK "IEC_Timer_0_DB_27"   // DB51
{ S7_Optimized_Access := 'TRUE' }
// stored: InstanceOfName IEC_TIMER, OfSystemLibElement IEC_TIMER, OfSystemLibVersion 1.0
"IEC_TIMER"
   // VAR
   //    PT : Time;
   //    ET { ExternalWritable := 'False'} : Time;
   //    IN : Bool;
   //    Q { ExternalWritable := 'False'} : Bool;
   // END_VAR
BEGIN
END_DATA_BLOCK

DATA_BLOCK "IEC_Timer_0_DB_28"   // DB52
{ S7_Optimized_Access := 'TRUE' }
// stored: InstanceOfName IEC_TIMER, OfSystemLibElement IEC_TIMER, OfSystemLibVersion 1.0
"IEC_TIMER"
   // VAR
   //    PT : Time;
   //    ET { ExternalWritable := 'False'} : Time;
   //    IN : Bool;
   //    Q { ExternalWritable := 'False'} : Bool;
   // END_VAR
BEGIN
END_DATA_BLOCK

DATA_BLOCK "IEC_Timer_0_DB_3"   // DB16
{ S7_Optimized_Access := 'TRUE' }
// stored: InstanceOfName IEC_TIMER, OfSystemLibElement IEC_TIMER, OfSystemLibVersion 1.0
"IEC_TIMER"
   // VAR
   //    PT : Time;
   //    ET { ExternalWritable := 'False'} : Time;
   //    IN : Bool;
   //    Q { ExternalWritable := 'False'} : Bool;
   // END_VAR
BEGIN
END_DATA_BLOCK

DATA_BLOCK "IEC_Timer_0_DB_30"   // DB54
{ S7_Optimized_Access := 'TRUE' }
// stored: InstanceOfName IEC_TIMER, OfSystemLibElement IEC_TIMER, OfSystemLibVersion 1.0
"IEC_TIMER"
   // VAR
   //    PT : Time;
   //    ET { ExternalWritable := 'False'} : Time;
   //    IN : Bool;
   //    Q { ExternalWritable := 'False'} : Bool;
   // END_VAR
BEGIN
END_DATA_BLOCK

DATA_BLOCK "IEC_Timer_0_DB_4"   // DB6
{ S7_Optimized_Access := 'TRUE' }
// stored: InstanceOfName IEC_TIMER, OfSystemLibElement IEC_TIMER, OfSystemLibVersion 1.0
"IEC_TIMER"
   // VAR
   //    PT : Time;
   //    ET { ExternalWritable := 'False'} : Time;
   //    IN : Bool;
   //    Q { ExternalWritable := 'False'} : Bool;
   // END_VAR
BEGIN
END_DATA_BLOCK

DATA_BLOCK "IEC_Timer_0_DB_5"   // DB18
{ S7_Optimized_Access := 'TRUE' }
// stored: InstanceOfName IEC_TIMER, OfSystemLibElement IEC_TIMER, OfSystemLibVersion 1.0
"IEC_TIMER"
   // VAR
   //    PT : Time;
   //    ET { ExternalWritable := 'False'} : Time;
   //    IN : Bool;
   //    Q { ExternalWritable := 'False'} : Bool;
   // END_VAR
BEGIN
END_DATA_BLOCK

DATA_BLOCK "IEC_Timer_0_DB_55"   // DB85
{ S7_Optimized_Access := 'TRUE' }
// stored: InstanceOfName IEC_TIMER, OfSystemLibElement IEC_TIMER, OfSystemLibVersion 1.0
"IEC_TIMER"
   // VAR
   //    PT : Time;
   //    ET { ExternalWritable := 'False'} : Time;
   //    IN : Bool;
   //    Q { ExternalWritable := 'False'} : Bool;
   // END_VAR
BEGIN
END_DATA_BLOCK

DATA_BLOCK "IEC_Timer_0_DB_7"   // DB46
{ S7_Optimized_Access := 'TRUE' }
// stored: InstanceOfName IEC_TIMER, OfSystemLibElement IEC_TIMER, OfSystemLibVersion 1.0
"IEC_TIMER"
   // VAR
   //    PT : Time;
   //    ET { ExternalWritable := 'False'} : Time;
   //    IN : Bool;
   //    Q { ExternalWritable := 'False'} : Bool;
   // END_VAR
BEGIN
END_DATA_BLOCK

DATA_BLOCK "IEC_Timer_0_DB_72"   // DB82
{ S7_Optimized_Access := 'TRUE' }
// stored: InstanceOfName IEC_TIMER, OfSystemLibElement IEC_TIMER, OfSystemLibVersion 1.0
"IEC_TIMER"
   // VAR
   //    PT : Time;
   //    ET { ExternalWritable := 'False'} : Time;
   //    IN : Bool;
   //    Q { ExternalWritable := 'False'} : Bool;
   // END_VAR
BEGIN
END_DATA_BLOCK

DATA_BLOCK "IEC_Timer_0_DB_73"   // DB93
{ S7_Optimized_Access := 'TRUE' }
// stored: InstanceOfName IEC_TIMER, OfSystemLibElement IEC_TIMER, OfSystemLibVersion 1.0
"IEC_TIMER"
   // VAR
   //    PT : Time;
   //    ET { ExternalWritable := 'False'} : Time;
   //    IN : Bool;
   //    Q { ExternalWritable := 'False'} : Bool;
   // END_VAR
BEGIN
END_DATA_BLOCK

DATA_BLOCK "IEC_Timer_0_DB_74"   // DB98
{ S7_Optimized_Access := 'TRUE' }
// stored: InstanceOfName IEC_TIMER, OfSystemLibElement IEC_TIMER, OfSystemLibVersion 1.0
"IEC_TIMER"
   // VAR
   //    PT : Time;
   //    ET { ExternalWritable := 'False'} : Time;
   //    IN : Bool;
   //    Q { ExternalWritable := 'False'} : Bool;
   // END_VAR
BEGIN
END_DATA_BLOCK

DATA_BLOCK "IEC_Timer_0_DB_75"   // DB102
{ S7_Optimized_Access := 'TRUE' }
// stored: InstanceOfName IEC_TIMER, OfSystemLibElement IEC_TIMER, OfSystemLibVersion 1.0
"IEC_TIMER"
   // VAR
   //    PT : Time;
   //    ET { ExternalWritable := 'False'} : Time;
   //    IN : Bool;
   //    Q { ExternalWritable := 'False'} : Bool;
   // END_VAR
BEGIN
END_DATA_BLOCK

DATA_BLOCK "IEC_Timer_0_DB_76"   // DB109
{ S7_Optimized_Access := 'TRUE' }
// stored: InstanceOfName IEC_TIMER, OfSystemLibElement IEC_TIMER, OfSystemLibVersion 1.0
"IEC_TIMER"
   // VAR
   //    PT : Time;
   //    ET { ExternalWritable := 'False'} : Time;
   //    IN : Bool;
   //    Q { ExternalWritable := 'False'} : Bool;
   // END_VAR
BEGIN
END_DATA_BLOCK

DATA_BLOCK "IEC_Timer_0_DB_77"   // DB113
{ S7_Optimized_Access := 'TRUE' }
// stored: InstanceOfName IEC_TIMER, OfSystemLibElement IEC_TIMER, OfSystemLibVersion 1.0
"IEC_TIMER"
   // VAR
   //    PT : Time;
   //    ET { ExternalWritable := 'False'} : Time;
   //    IN : Bool;
   //    Q { ExternalWritable := 'False'} : Bool;
   // END_VAR
BEGIN
END_DATA_BLOCK

DATA_BLOCK "IEC_Timer_0_DB_78"   // DB114
{ S7_Optimized_Access := 'TRUE' }
// stored: InstanceOfName IEC_TIMER, OfSystemLibElement IEC_TIMER, OfSystemLibVersion 1.0
"IEC_TIMER"
   // VAR
   //    PT : Time;
   //    ET { ExternalWritable := 'False'} : Time;
   //    IN : Bool;
   //    Q { ExternalWritable := 'False'} : Bool;
   // END_VAR
BEGIN
END_DATA_BLOCK

DATA_BLOCK "IEC_Timer_0_DB_8"   // DB25
{ S7_Optimized_Access := 'TRUE' }
// stored: InstanceOfName IEC_TIMER, OfSystemLibElement IEC_TIMER, OfSystemLibVersion 1.0
"IEC_TIMER"
   // VAR
   //    PT : Time;
   //    ET { ExternalWritable := 'False'} : Time;
   //    IN : Bool;
   //    Q { ExternalWritable := 'False'} : Bool;
   // END_VAR
BEGIN
END_DATA_BLOCK

DATA_BLOCK "IEC_Timer_0_DB_9"   // DB26
{ S7_Optimized_Access := 'TRUE' }
// stored: InstanceOfName IEC_TIMER, OfSystemLibElement IEC_TIMER, OfSystemLibVersion 1.0
"IEC_TIMER"
   // VAR
   //    PT : Time;
   //    ET { ExternalWritable := 'False'} : Time;
   //    IN : Bool;
   //    Q { ExternalWritable := 'False'} : Bool;
   // END_VAR
BEGIN
END_DATA_BLOCK
